// Mitsubishi GX Works2 project: ex02   PLC: Q02/Q02H

PROGRAM MAIN
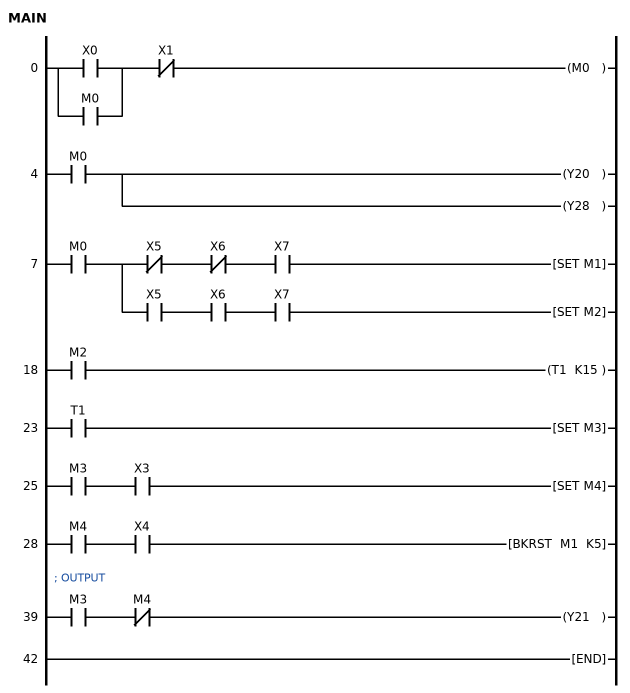
0     LD      X0
      OR      M0
      ANI     X1
      OUT     M0
4     LD      M0
      OUT     Y20
      OUT     Y28
7     LD      M0
      MPS
      ANI     X5
      ANI     X6
      AND     X7
      SET     M1
      MPP
      AND     X5
      AND     X6
      AND     X7
      SET     M2
18    LD      M2
      OUT     T1 K15
23    LD      T1
      SET     M3
25    LD      M3
      AND     X3
      SET     M4
28    LD      M4
      AND     X4
      BKRST   M1 K5
; OUTPUT
39    LD      M3
      ANI     M4
      OUT     Y21
42    END
END_PROGRAM
